Staubli VAL3: moveX.pgx

public program moveX(num nDx (dimensions=1))
  local point pFinal
  local point pHere
begin
  //pHere=here(tActive,frActive)
  //pFinal=compose(pHere,frActive,{nDx,0,0,0,0,0})
  pDest=compose(pDest,frActive,{nDx,0,0,0,0,0})
  //movel(pFinal,tActive,mNomSpeed)
  movel(pDest,tActive,mNomSpeed)
end
